// TIA Portal V17 export
// export: Created 2023-04-03T06:31:28.3544306Z, ExportSetting WithDefaults, DisplayName Totally Integrated Automation Portal, DisplayVersion V17 Update 4, DisplayName TIA Portal Openness, DisplayVersion V17 Update 4, DisplayName TIA Portal Version Control Interface, DisplayVersion V17, DisplayName STEP 7 Professional, DisplayVersion V17 Update 4, DisplayName STEP 7 Safety, DisplayVersion V17, DisplayName WinCC Professional, DisplayVersion V17 Update 4
DATA_BLOCK "MvSkid_2"   // DB46
{ S7_Optimized_Access := 'TRUE' }
VERSION : 0.1
// stored: AutoNumber true, DBAccessibleFromOPCUA true, DBAccessibleFromWebserver true, IsOnlyStoredInLoadMemory false, IsRetainMemResEnabled false, IsWriteProtectedInAS false, MemoryReserve 100
   VAR RETAIN
      TCON { S7_SetPoint := 'True'} : TCON_IP_v4;
   END_VAR
   VAR
      arrData : Array[1..125] of Word;
      xREQ : Bool;
      iCountDone : Int := 1;
      iCountRead : Int := 1;
      MBmode : USInt;
      MBdataAddr : UDInt;
      MBdataLen : UInt;
      R : "R_MV";
      W { S7_SetPoint := 'True'} : "W_MV";
      xFltSt { S7_SetPoint := 'True'} : Bool;
      xAlmSt : Bool;
      xWarnSt : Bool;
      wLine1DiscSt : Word;
      wLine2DiscSt : Word;
      wProt1DiscSt : Word;
      wProt1CircBrkSt : Word;
   END_VAR
BEGIN
   TCON.RemoteAddress.ADDR[1] := 192;
   TCON.RemoteAddress.ADDR[2] := 168;
   TCON.RemoteAddress.ADDR[3] := 150;
   TCON.RemoteAddress.ADDR[4] := 44;
END_DATA_BLOCK
